Fanuc KAREL source: ATT_WINDOW_D.kl

PROGRAM T
%NOLOCKGROUP
VAR
 v0 : STRING[40]
 v1 : STRING[40]
 v2 : INTEGER
 v3 : INTEGER
 v4 : STRING[40]
 v5 : INTEGER
BEGIN
 ATT_WINDOW_D(v0, v1, v2, v3, v4, v5)
END T
